TYPE ST_TBOT_TC_SubLevelEAP :
STRUCT
	bTCDwrSafeToMoveEAP (*AT %I**): BOOL:=TRUE;
	
	//ipTCDrawerCylExtendRS_EAP	(*AT %Q**): BOOL;		
	//ipTCDrawerCylRetractRS_EAP	(*AT %Q**): BOOL;	
END_STRUCT
END_TYPE

(* stored: Version 1.1.0.1, ProductVersion 3.1.4022.18
   DUT ST_TBOT_TC_SubLevelEAP: Id {97672cf1-6d21-4b57-a8cf-628cd34e603e} *)
